{attribute 'qualified_only'}
VAR_GLOBAL
END_VAR

(* stored: Version 1.1.0.1, ProductVersion 3.1.4022.7
   GVL GVL_02_Parameter_Servo_Motor_Shelf_C: Id {022bbaa7-77df-47fb-9db5-84d14be65d79} *)
